(* Logix 5000 project; controller Sucrose_Main Emulate 5570 rev 20.12; software revision 20.01; part 29 of 30 *)
(* tags used below, declared in another part *)
   Alarm_ACK_Master_Timer : TIMER;
   DI_E23_3 : ALIAS FOR FLX_E23:3:I;   // Discrete Input EN2T_FLX 192.168.1.23
   DO_E24_3 : ALIAS FOR FLX_E24:3:O;   // Discrete Output EN2T_FLX 192.168.1.24
   DO_E24_4 : ALIAS FOR FLX_E24:4:O;   // Discrete Output EN2T_FLX 192.168.1.24
   DO_E24_5 : ALIAS FOR FLX_E24:5:O;   // Discrete Output EN2T_FLX 192.168.1.24
   FV230202_AOI : QSI_Flow_Valve;   // FV-23-02-02 SUCROSE TANK #2 INLET/SPRAYBALL VALVE
   FV230302_AOI : QSI_Flow_Valve;   // FV-23-03-02 SUCROSE TANK #3 INLET/SPRAYBALL VALVE
   FV751201_AOI : QSI_Flow_Valve;   // FV-75-12-01 SUCROSE TANK #2 BLANKETING STEAM TRAP ISOLATION VALVE
   FV751301_AOI : QSI_Flow_Valve;   // FV-75-13-01 SUCROSE TANK #3 BLANKETING STEAM TRAP ISOLATION VALVE
   FV931102_AOI : QSI_Flow_Valve;
   FV931103_AOI : QSI_Flow_Valve;
   FV931201_AOI : QSI_Flow_Valve;   // FV-93-12-01 STERILE AIR FLT-93-12-01 SHUT OFF VALVE
   FV931202_AOI : QSI_Flow_Valve;
   FV931203_AOI : QSI_Flow_Valve;
   FV931301_AOI : QSI_Flow_Valve;   // FV-93-13-01 STERILE AIR FLT-93-13-01 SHUT OFF VALVE
   FV931302_AOI : QSI_Flow_Valve;
   FV931303_AOI : QSI_Flow_Valve;
   HTR760101_AOI : QSI_Discrete_Device;   // HTR-76-01-01 SUCROSE TANK #1 UTILITY HOT WATER ELECTRIC HEATER ENABLE
   Sucrose_MM_Enable : BOOL;
   SucroseCIP_TK230201_REMOTE : CIP_REMOTE;
   SucroseCIP_TK230301_REMOTE : CIP_REMOTE;
   SucroseTanks : Area_Program;
(* TanksArea_EN2T_IO_Discrete_DO_E24_3, continued *)

ROUTINE _04_FV230202   (* ladder *)
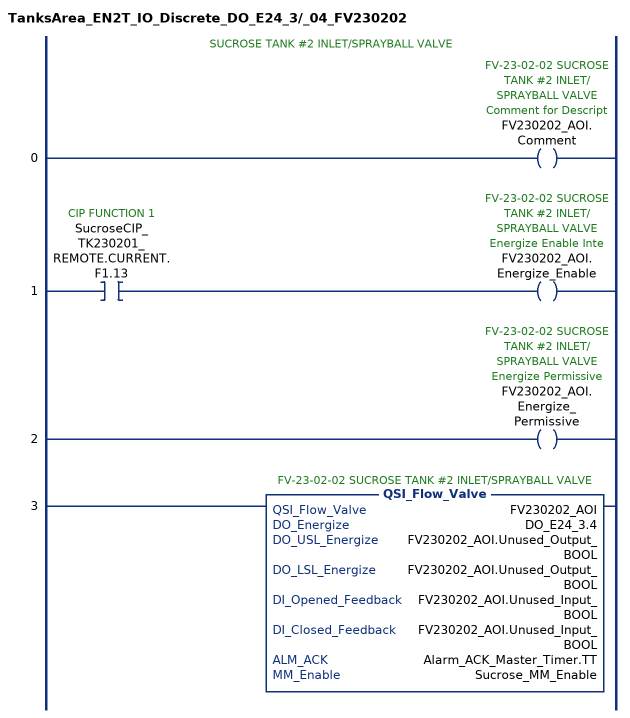
   // SUCROSE TANK #2 INLET/SPRAYBALL VALVE
   0: OTE(FV230202_AOI.Comment);
   1: XIC(SucroseCIP_TK230201_REMOTE.CURRENT.F1.13)OTE(FV230202_AOI.Energize_Enable);
   2: OTE(FV230202_AOI.Energize_Permissive);
   3: QSI_Flow_Valve(FV230202_AOI,DO_E24_3.4,FV230202_AOI.Unused_Output_BOOL,FV230202_AOI.Unused_Output_BOOL,FV230202_AOI.Unused_Input_BOOL,FV230202_AOI.Unused_Input_BOOL,Alarm_ACK_Master_Timer.TT,Sucrose_MM_Enable);
END_ROUTINE

ROUTINE _06_FV751201   (* ladder *)
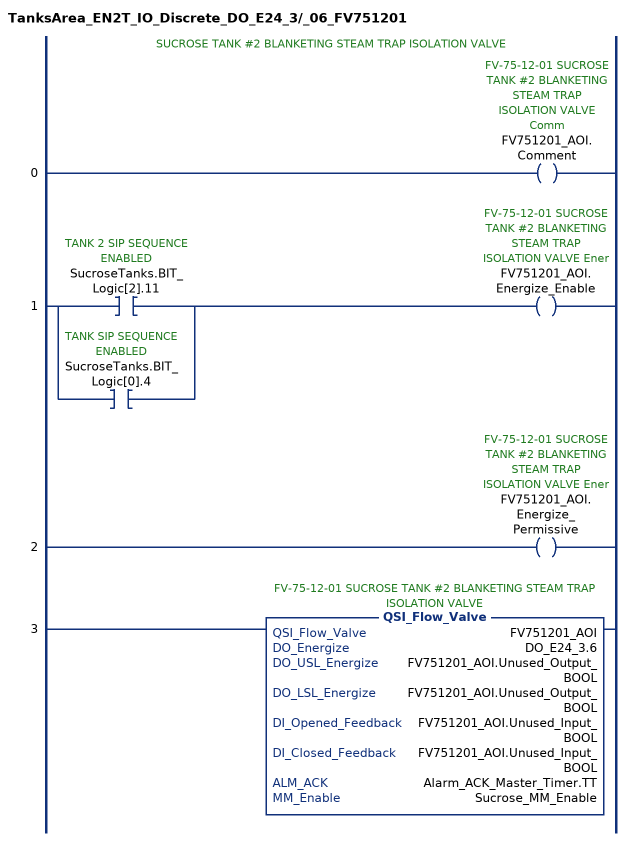
   // SUCROSE TANK #2 BLANKETING STEAM TRAP ISOLATION VALVE
   0: OTE(FV751201_AOI.Comment);
   1: [XIC(SucroseTanks.BIT_Logic[2].11) ,XIC(SucroseTanks.BIT_Logic[0].4) ]OTE(FV751201_AOI.Energize_Enable);
   2: OTE(FV751201_AOI.Energize_Permissive);
   3: QSI_Flow_Valve(FV751201_AOI,DO_E24_3.6,FV751201_AOI.Unused_Output_BOOL,FV751201_AOI.Unused_Output_BOOL,FV751201_AOI.Unused_Input_BOOL,FV751201_AOI.Unused_Input_BOOL,Alarm_ACK_Master_Timer.TT,Sucrose_MM_Enable);
END_ROUTINE

ROUTINE _07_FV931201   (* ladder *)
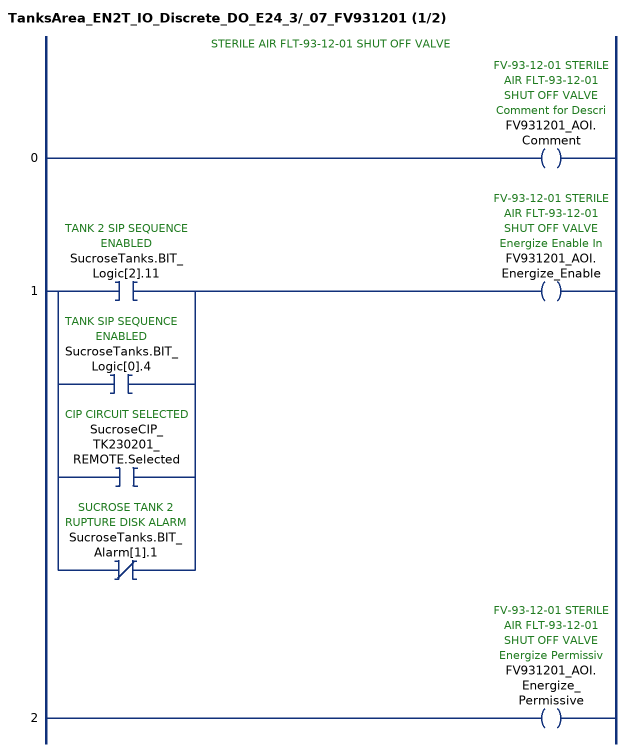
   // STERILE AIR FLT-93-12-01 SHUT OFF VALVE
   0: OTE(FV931201_AOI.Comment);
   1: [XIC(SucroseTanks.BIT_Logic[2].11) ,XIC(SucroseTanks.BIT_Logic[0].4) ,XIC(SucroseCIP_TK230201_REMOTE.Selected) ,XIO(SucroseTanks.BIT_Alarm[1].1) ]OTE(FV931201_AOI.Energize_Enable);
   2: OTE(FV931201_AOI.Energize_Permissive);
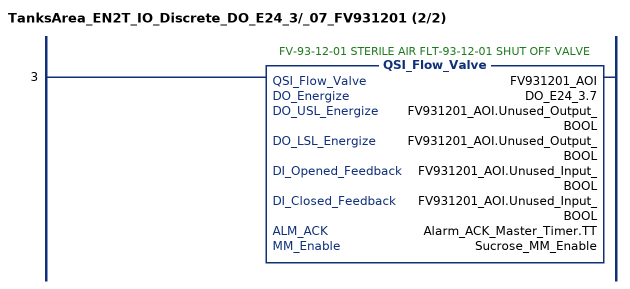
   3: QSI_Flow_Valve(FV931201_AOI,DO_E24_3.7,FV931201_AOI.Unused_Output_BOOL,FV931201_AOI.Unused_Output_BOOL,FV931201_AOI.Unused_Input_BOOL,FV931201_AOI.Unused_Input_BOOL,Alarm_ACK_Master_Timer.TT,Sucrose_MM_Enable);
END_ROUTINE

ROUTINE _08_FV931102   (* ladder *)
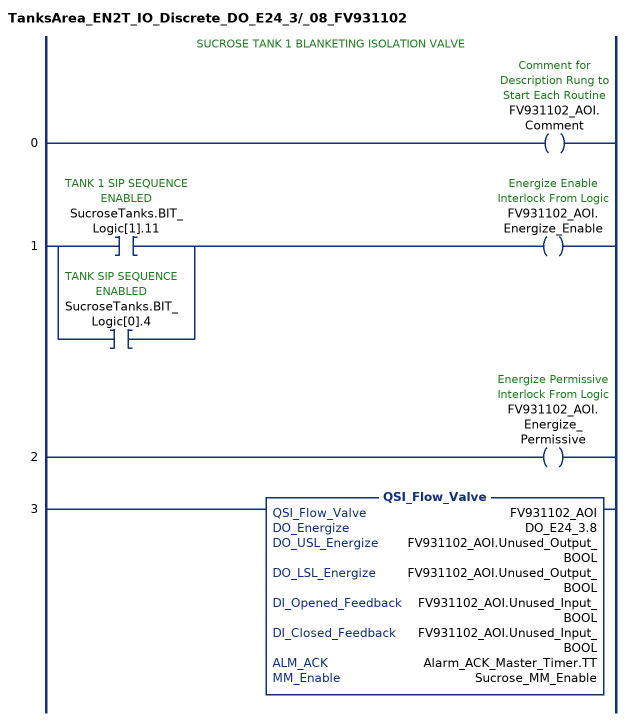
   // SUCROSE TANK 1 BLANKETING ISOLATION VALVE
   0: OTE(FV931102_AOI.Comment);
   1: [XIC(SucroseTanks.BIT_Logic[1].11) ,XIC(SucroseTanks.BIT_Logic[0].4) ]OTE(FV931102_AOI.Energize_Enable);
   2: OTE(FV931102_AOI.Energize_Permissive);
   3: QSI_Flow_Valve(FV931102_AOI,DO_E24_3.8,FV931102_AOI.Unused_Output_BOOL,FV931102_AOI.Unused_Output_BOOL,FV931102_AOI.Unused_Input_BOOL,FV931102_AOI.Unused_Input_BOOL,Alarm_ACK_Master_Timer.TT,Sucrose_MM_Enable);
END_ROUTINE

ROUTINE _09_FV931103   (* ladder *)
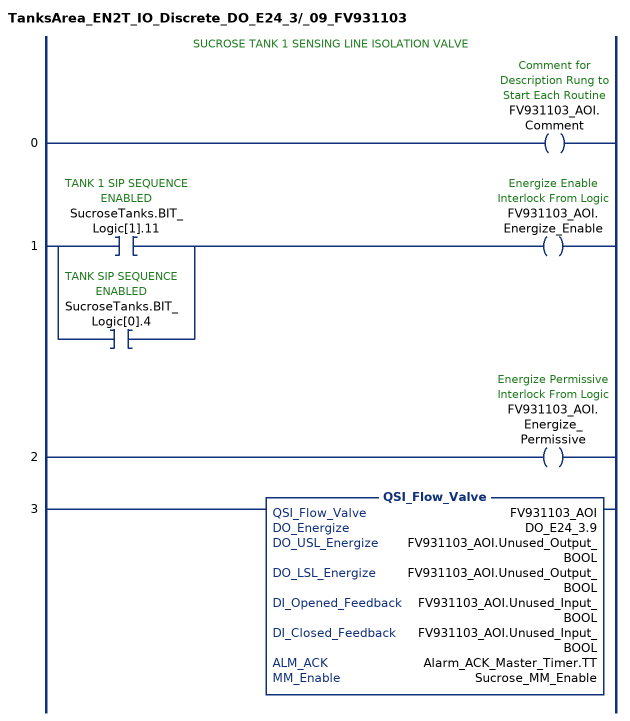
   // SUCROSE TANK 1 SENSING LINE ISOLATION VALVE
   0: OTE(FV931103_AOI.Comment);
   1: [XIC(SucroseTanks.BIT_Logic[1].11) ,XIC(SucroseTanks.BIT_Logic[0].4) ]OTE(FV931103_AOI.Energize_Enable);
   2: OTE(FV931103_AOI.Energize_Permissive);
   3: QSI_Flow_Valve(FV931103_AOI,DO_E24_3.9,FV931103_AOI.Unused_Output_BOOL,FV931103_AOI.Unused_Output_BOOL,FV931103_AOI.Unused_Input_BOOL,FV931103_AOI.Unused_Input_BOOL,Alarm_ACK_Master_Timer.TT,Sucrose_MM_Enable);
END_ROUTINE

ROUTINE _10_FV230302   (* ladder *)
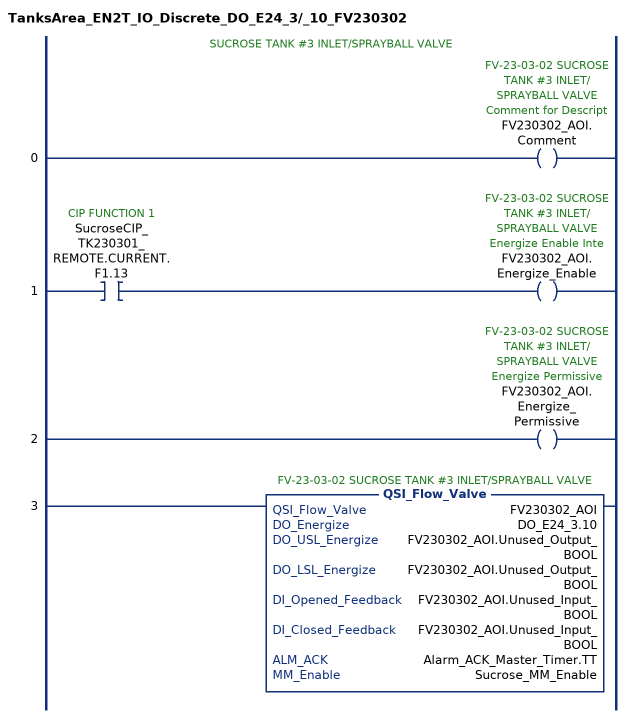
   // SUCROSE TANK #3 INLET/SPRAYBALL VALVE
   0: OTE(FV230302_AOI.Comment);
   1: XIC(SucroseCIP_TK230301_REMOTE.CURRENT.F1.13)OTE(FV230302_AOI.Energize_Enable);
   2: OTE(FV230302_AOI.Energize_Permissive);
   3: QSI_Flow_Valve(FV230302_AOI,DO_E24_3.10,FV230302_AOI.Unused_Output_BOOL,FV230302_AOI.Unused_Output_BOOL,FV230302_AOI.Unused_Input_BOOL,FV230302_AOI.Unused_Input_BOOL,Alarm_ACK_Master_Timer.TT,Sucrose_MM_Enable);
END_ROUTINE

ROUTINE _12_FV751301   (* ladder *)
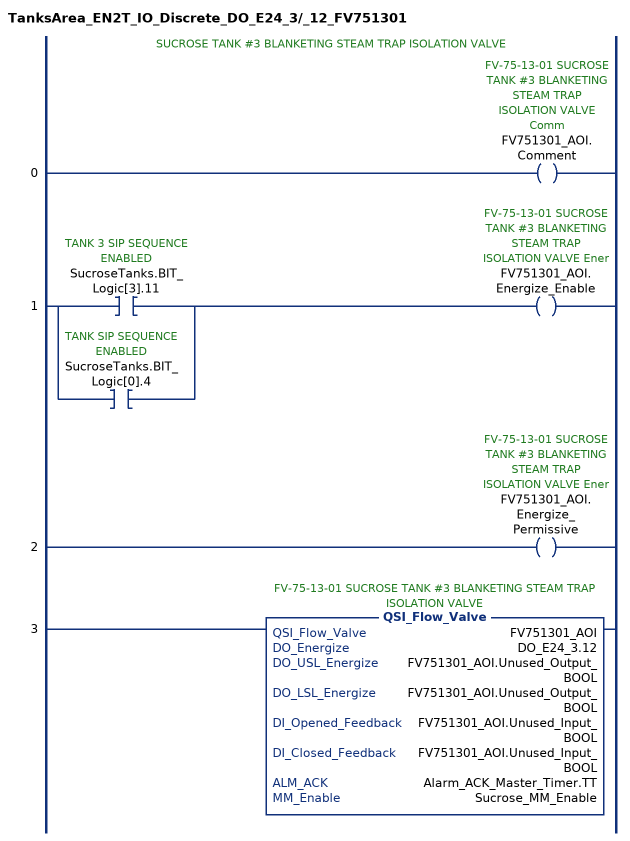
   // SUCROSE TANK #3 BLANKETING STEAM TRAP ISOLATION VALVE
   0: OTE(FV751301_AOI.Comment);
   1: [XIC(SucroseTanks.BIT_Logic[3].11) ,XIC(SucroseTanks.BIT_Logic[0].4) ]OTE(FV751301_AOI.Energize_Enable);
   2: OTE(FV751301_AOI.Energize_Permissive);
   3: QSI_Flow_Valve(FV751301_AOI,DO_E24_3.12,FV751301_AOI.Unused_Output_BOOL,FV751301_AOI.Unused_Output_BOOL,FV751301_AOI.Unused_Input_BOOL,FV751301_AOI.Unused_Input_BOOL,Alarm_ACK_Master_Timer.TT,Sucrose_MM_Enable);
END_ROUTINE

ROUTINE _13_FV931301   (* ladder *)
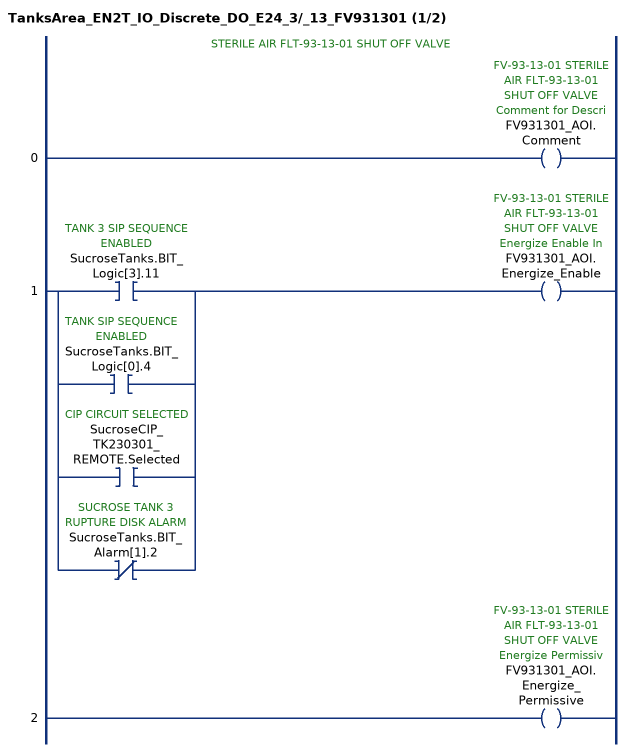
   // STERILE AIR FLT-93-13-01 SHUT OFF VALVE
   0: OTE(FV931301_AOI.Comment);
   1: [XIC(SucroseTanks.BIT_Logic[3].11) ,XIC(SucroseTanks.BIT_Logic[0].4) ,XIC(SucroseCIP_TK230301_REMOTE.Selected) ,XIO(SucroseTanks.BIT_Alarm[1].2) ]OTE(FV931301_AOI.Energize_Enable);
   2: OTE(FV931301_AOI.Energize_Permissive);
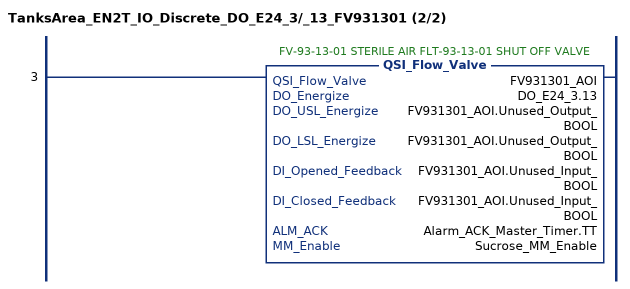
   3: QSI_Flow_Valve(FV931301_AOI,DO_E24_3.13,FV931301_AOI.Unused_Output_BOOL,FV931301_AOI.Unused_Output_BOOL,FV931301_AOI.Unused_Input_BOOL,FV931301_AOI.Unused_Input_BOOL,Alarm_ACK_Master_Timer.TT,Sucrose_MM_Enable);
END_ROUTINE

ROUTINE MainRoutine   (* ladder *)
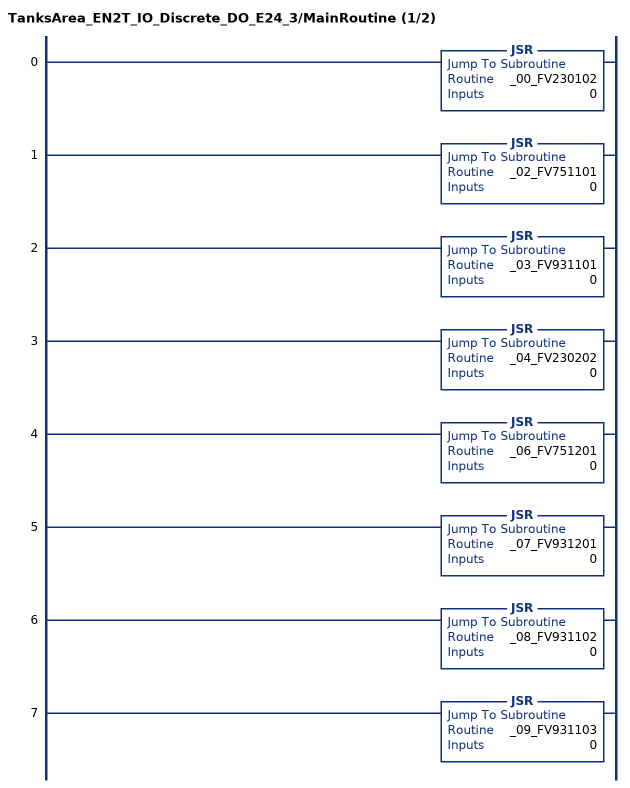
   0: JSR(_00_FV230102,0);
   1: JSR(_02_FV751101,0);
   2: JSR(_03_FV931101,0);
   3: JSR(_04_FV230202,0);
   4: JSR(_06_FV751201,0);
   5: JSR(_07_FV931201,0);
   6: JSR(_08_FV931102,0);
   7: JSR(_09_FV931103,0);
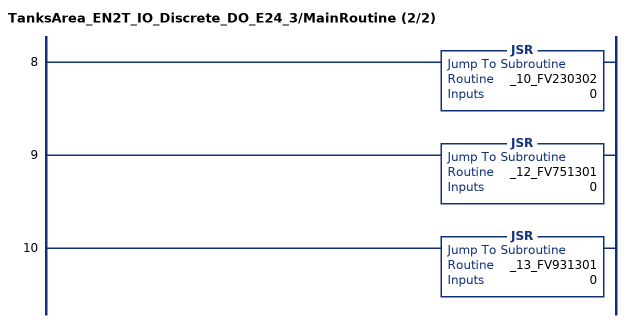
   8: JSR(_10_FV230302,0);
   9: JSR(_12_FV751301,0);
   10: JSR(_13_FV931301,0);
END_ROUTINE
END_PROGRAM

PROGRAM TanksArea_EN2T_IO_Discrete_DO_E24_4   (* main routine MainRoutine *)

ROUTINE _01_FV931202   (* ladder *)
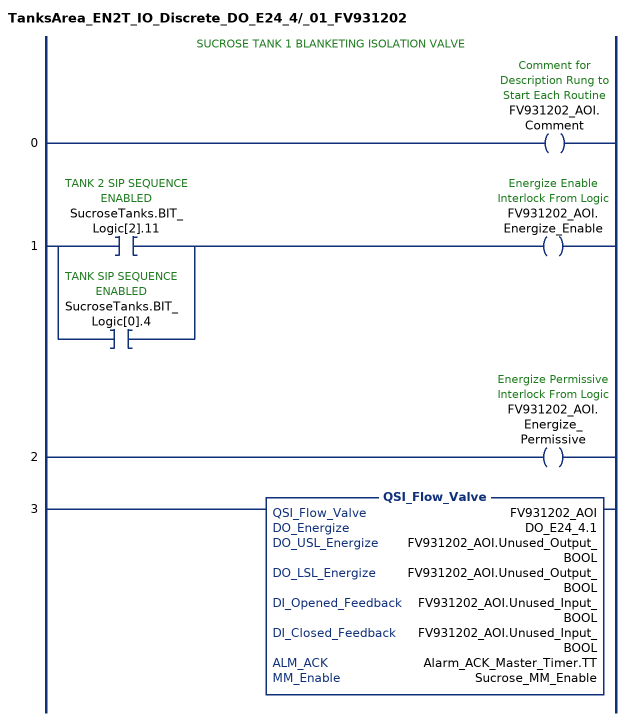
   // SUCROSE TANK 1 BLANKETING ISOLATION VALVE
   0: OTE(FV931202_AOI.Comment);
   1: [XIC(SucroseTanks.BIT_Logic[2].11) ,XIC(SucroseTanks.BIT_Logic[0].4) ]OTE(FV931202_AOI.Energize_Enable);
   2: OTE(FV931202_AOI.Energize_Permissive);
   3: QSI_Flow_Valve(FV931202_AOI,DO_E24_4.1,FV931202_AOI.Unused_Output_BOOL,FV931202_AOI.Unused_Output_BOOL,FV931202_AOI.Unused_Input_BOOL,FV931202_AOI.Unused_Input_BOOL,Alarm_ACK_Master_Timer.TT,Sucrose_MM_Enable);
END_ROUTINE

ROUTINE _02_FV931203   (* ladder *)
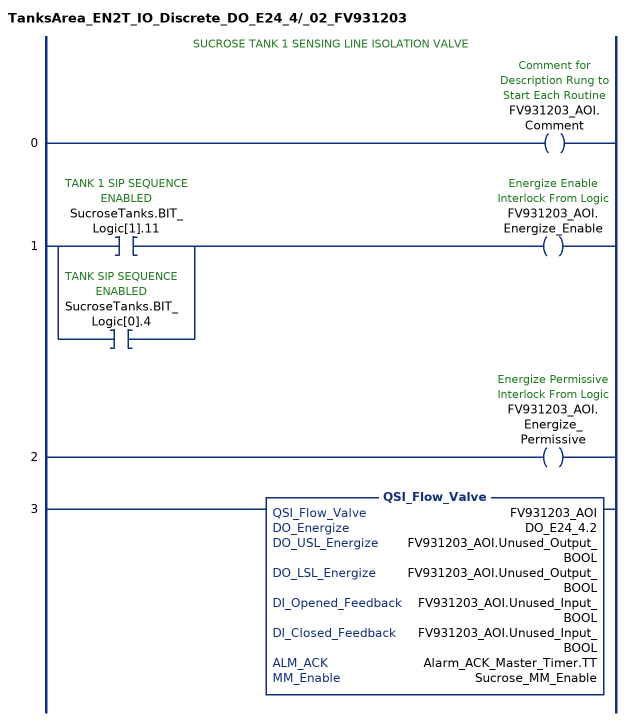
   // SUCROSE TANK 1 SENSING LINE ISOLATION VALVE
   0: OTE(FV931203_AOI.Comment);
   1: [XIC(SucroseTanks.BIT_Logic[1].11) ,XIC(SucroseTanks.BIT_Logic[0].4) ]OTE(FV931203_AOI.Energize_Enable);
   2: OTE(FV931203_AOI.Energize_Permissive);
   3: QSI_Flow_Valve(FV931203_AOI,DO_E24_4.2,FV931203_AOI.Unused_Output_BOOL,FV931203_AOI.Unused_Output_BOOL,FV931203_AOI.Unused_Input_BOOL,FV931203_AOI.Unused_Input_BOOL,Alarm_ACK_Master_Timer.TT,Sucrose_MM_Enable);
END_ROUTINE

ROUTINE _03_FV931302   (* ladder *)
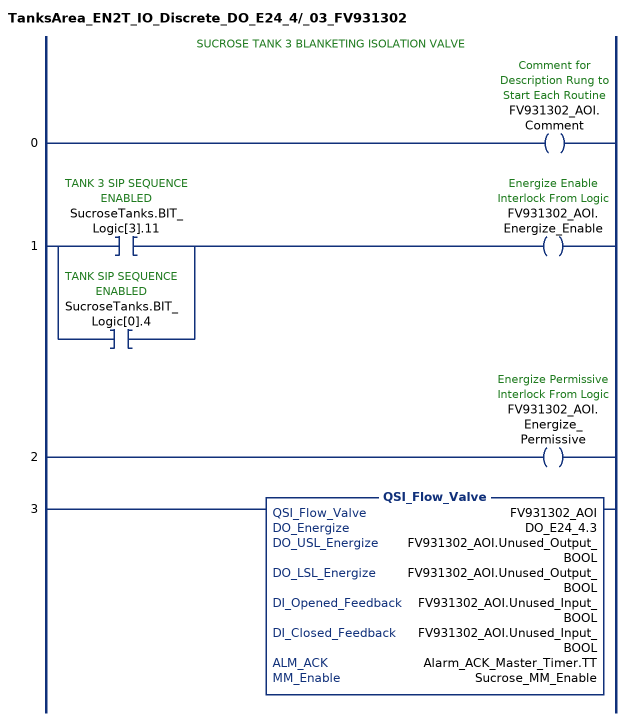
   // SUCROSE TANK 3 BLANKETING ISOLATION VALVE
   0: OTE(FV931302_AOI.Comment);
   1: [XIC(SucroseTanks.BIT_Logic[3].11) ,XIC(SucroseTanks.BIT_Logic[0].4) ]OTE(FV931302_AOI.Energize_Enable);
   2: OTE(FV931302_AOI.Energize_Permissive);
   3: QSI_Flow_Valve(FV931302_AOI,DO_E24_4.3,FV931302_AOI.Unused_Output_BOOL,FV931302_AOI.Unused_Output_BOOL,FV931302_AOI.Unused_Input_BOOL,FV931302_AOI.Unused_Input_BOOL,Alarm_ACK_Master_Timer.TT,Sucrose_MM_Enable);
END_ROUTINE

ROUTINE _06_FV931303   (* ladder *)
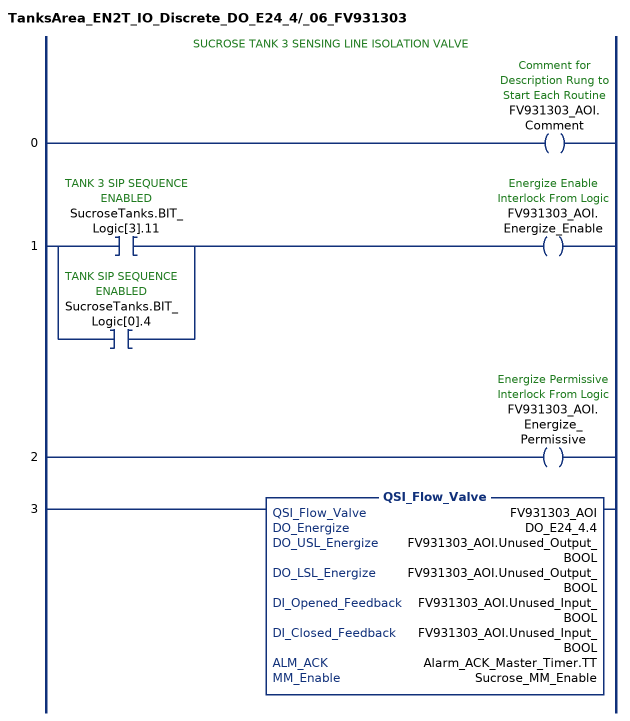
   // SUCROSE TANK 3 SENSING LINE ISOLATION VALVE
   0: OTE(FV931303_AOI.Comment);
   1: [XIC(SucroseTanks.BIT_Logic[3].11) ,XIC(SucroseTanks.BIT_Logic[0].4) ]OTE(FV931303_AOI.Energize_Enable);
   2: OTE(FV931303_AOI.Energize_Permissive);
   3: QSI_Flow_Valve(FV931303_AOI,DO_E24_4.4,FV931303_AOI.Unused_Output_BOOL,FV931303_AOI.Unused_Output_BOOL,FV931303_AOI.Unused_Input_BOOL,FV931303_AOI.Unused_Input_BOOL,Alarm_ACK_Master_Timer.TT,Sucrose_MM_Enable);
END_ROUTINE

ROUTINE MainRoutine   (* ladder *)
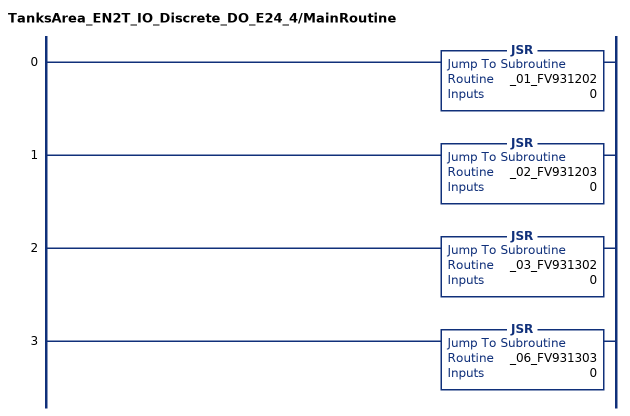
   0: JSR(_01_FV931202,0);
   1: JSR(_02_FV931203,0);
   2: JSR(_03_FV931302,0);
   3: JSR(_06_FV931303,0);
END_ROUTINE
END_PROGRAM

PROGRAM TanksArea_EN2T_IO_Discrete_DO_E24_5   (* main routine MainRoutine *)

ROUTINE _00_HTR760101   (* ladder *)
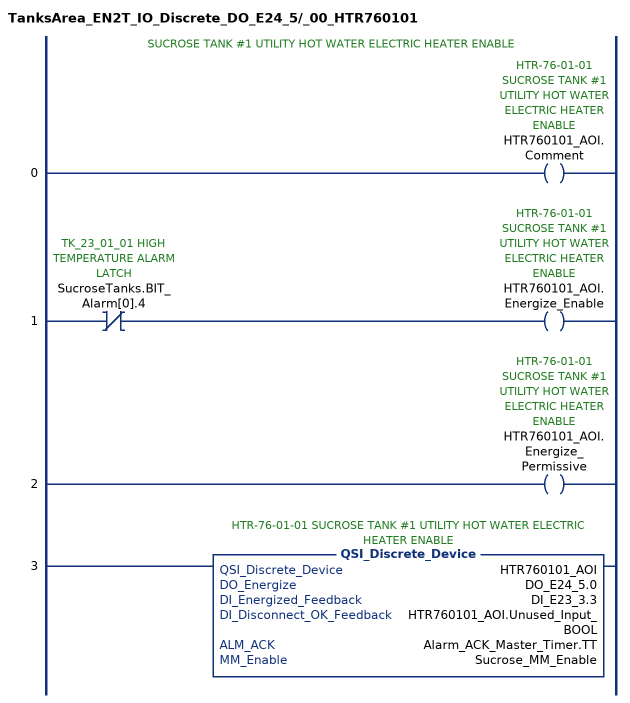
   // SUCROSE TANK #1 UTILITY HOT WATER ELECTRIC HEATER ENABLE
   0: OTE(HTR760101_AOI.Comment);
   1: XIO(SucroseTanks.BIT_Alarm[0].4)OTE(HTR760101_AOI.Energize_Enable);
   2: OTE(HTR760101_AOI.Energize_Permissive);
   3: QSI_Discrete_Device(HTR760101_AOI,DO_E24_5.0,DI_E23_3.3,HTR760101_AOI.Unused_Input_BOOL,Alarm_ACK_Master_Timer.TT,Sucrose_MM_Enable);
END_ROUTINE
